% RSLogix 500 project I2A JOB 12 B- MITCH_BAK034.RSS, saved by version 10.00.00.00 %
PROJECT "ML01B"    % processor: Bul.1763 MicroLogix 1100 Series B %

PROGRAM FILES
  LAD 2   11 rungs

DATA FILES
  O0 OUTPUT  4 elements
  I1 INPUT  6 elements
  S2 STATUS  66 elements
  B3 BINARY  1 elements
  T4 TIMER  1 elements
  C5 COUNTER  1 elements
  R6 CONTROL  1 elements
  N7 INTEGER  1 elements
  F8 FLOAT  1 elements

LADDER 2
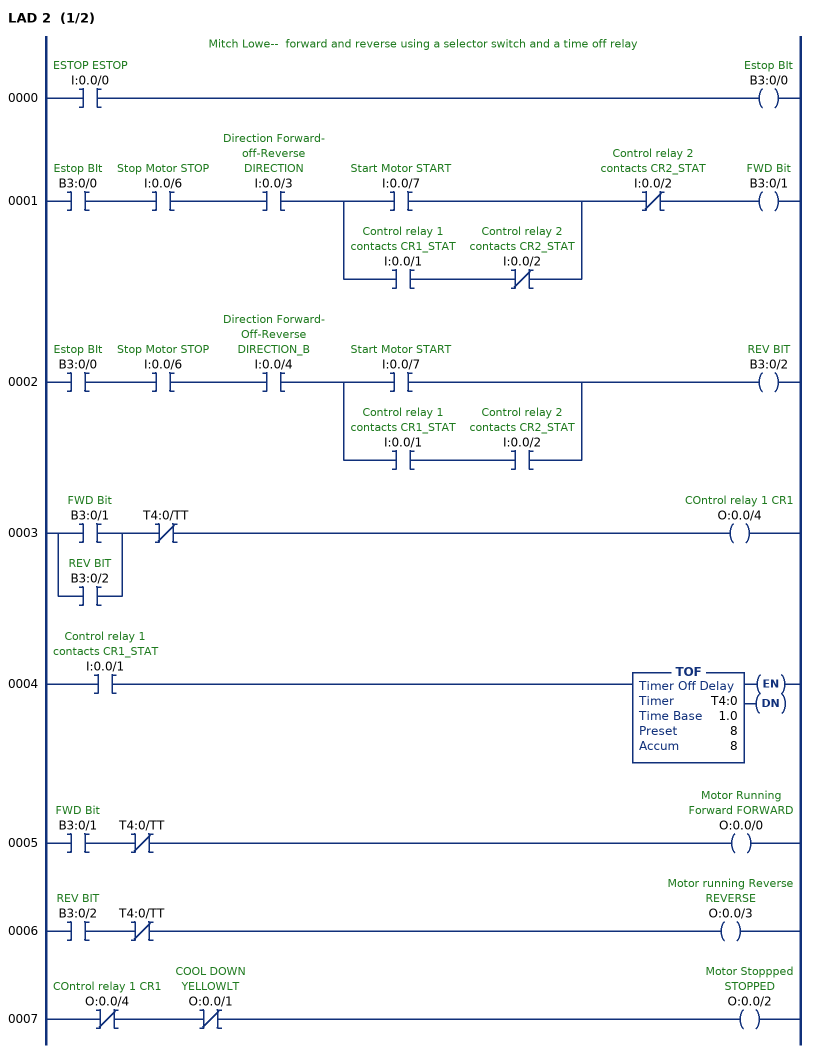
% Rung: 0 %
% Mitch Lowe--  forward and reverse using a selector switch and a time off relay %
SOR XIC I:0.0/0 OTE B3:0/0 EOR
%   I:0.0/0  ESTOP  "ESTOP" %
%   B3:0/0  "Estop BIt" %
% Rung: 1 %
SOR XIC B3:0/0 XIC I:0.0/6 XIC I:0.0/3 BST XIC I:0.0/7 NXB XIC I:0.0/1 XIO I:0.0/2 BND XIO I:0.0/2 OTE B3:0/1 EOR
%   B3:0/0  "Estop BIt" %
%   I:0.0/6  STOP  "Stop Motor" %
%   I:0.0/3  DIRECTION  "Direction Forward- off-Reverse" %
%   I:0.0/7  START  "Start Motor" %
%   I:0.0/1  CR1_STAT  "Control relay 1 contacts" %
%   I:0.0/2  CR2_STAT  "Control relay 2 contacts" %
%   B3:0/1  "FWD Bit" %
% Rung: 2 %
SOR XIC B3:0/0 XIC I:0.0/6 XIC I:0.0/4 BST XIC I:0.0/7 NXB XIC I:0.0/1 XIC I:0.0/2 BND OTE B3:0/2 EOR
%   B3:0/0  "Estop BIt" %
%   I:0.0/6  STOP  "Stop Motor" %
%   I:0.0/4  DIRECTION_B  "Direction Forward- Off-Reverse" %
%   I:0.0/7  START  "Start Motor" %
%   I:0.0/1  CR1_STAT  "Control relay 1 contacts" %
%   I:0.0/2  CR2_STAT  "Control relay 2 contacts" %
%   B3:0/2  "REV BIT" %
% Rung: 3 %
SOR BST XIC B3:0/1 NXB XIC B3:0/2 BND XIO T4:0/TT OTE O:0.0/4 EOR
%   B3:0/1  "FWD Bit" %
%   B3:0/2  "REV BIT" %
%   O:0.0/4  CR1  "COntrol relay 1" %
% Rung: 4 %
SOR XIC I:0.0/1 TOF T4:0 1.0 8 8 EOR
%   I:0.0/1  CR1_STAT  "Control relay 1 contacts" %
% Rung: 5 %
SOR XIC B3:0/1 XIO T4:0/TT OTE O:0.0/0 EOR
%   B3:0/1  "FWD Bit" %
%   O:0.0/0  FORWARD  "Motor Running Forward" %
% Rung: 6 %
SOR XIC B3:0/2 XIO T4:0/TT OTE O:0.0/3 EOR
%   B3:0/2  "REV BIT" %
%   O:0.0/3  REVERSE  "Motor running Reverse" %
% Rung: 7 %
SOR XIO O:0.0/4 XIO O:0.0/1 OTE O:0.0/2 EOR
%   O:0.0/4  CR1  "COntrol relay 1" %
%   O:0.0/1  YELLOWLT  "COOL DOWN" %
%   O:0.0/2  STOPPED  "Motor Stoppped" %

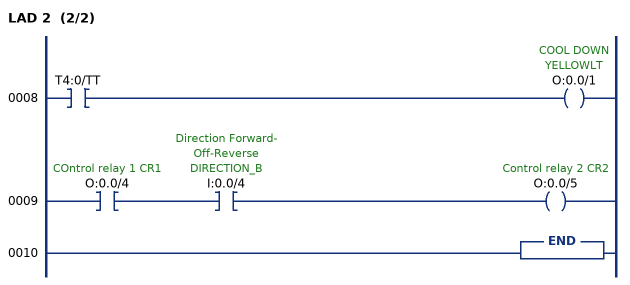
% Rung: 8 %
SOR XIC T4:0/TT OTE O:0.0/1 EOR
%   O:0.0/1  YELLOWLT  "COOL DOWN" %
% Rung: 9 %
SOR XIC O:0.0/4 XIC I:0.0/4 OTE O:0.0/5 EOR
%   O:0.0/4  CR1  "COntrol relay 1" %
%   I:0.0/4  DIRECTION_B  "Direction Forward- Off-Reverse" %
%   O:0.0/5  CR2  "Control relay 2" %
% Rung: 10 %
SOR END EOR

OTHER DOCUMENTED ADDRESSES
  I:0.0/5  2PSSA  "2 position selector switch A"
  I:0.0/8  PB3  "N.O pushbutton"

DATA TABLE (non-zero values as saved)
DATA B3
% B3:0 % 0X0001
DATA T4
% .PRE .ACC %
% T4:0 % 8 8
